{attribute 'qualified_only'}
{attribute 'strict'}
TYPE E_TunePreSets :
(
	Fast := 0, 	// Fast settling with overshoots of 10%-20%
	Slow,		// Slower settling with low overshoot
	Asymptotic	//Almost asymptotic settling with extremely small overshoot
);
END_TYPE

(* stored: Version 1.1.0.1, ProductVersion 3.1.4024.11
   DUT E_TunePreSets: Id {edc58d97-2ead-070e-37dd-b2e8dd391050} *)
